// TIA Portal V16 export
// export: Created 2025-07-26T13:20:06.7071257Z, ExportSetting WithDefaults, DisplayName Totally Integrated Automation Portal, DisplayVersion V16, DisplayName TIA Portal Version Control Interface, DisplayVersion V16, DisplayName TIA Portal Openness, DisplayVersion V16, DisplayName STEP 7 Professional, DisplayVersion V16, DisplayName STEP 7 Safety, DisplayVersion V16, DisplayName WinCC Advanced, DisplayVersion V16
VAR_GLOBAL   // PLC tag table "Tag table_1"
END_VAR
